FUNCTION_BLOCK M_ADD (* Add two matrices of REAL *)
  (* Standard: 61499-1 *)
  (* Version 0.2, 2007-10-24, JHC, Holobloc Inc, Changed RHS of sequences to MATRIX. *)
  (* Version 0.1, 2007-10-19, JHC, Holobloc Inc, Moved to fb.rt.math.matrix. *)
  (* Version 0.0, 2002-03-05, JHC, Rockwell Automation *)
  (* Compiler header: package fb.rt.math.matrix; *)
  (* Compiler Java Sun JDK 1.6.0 *)
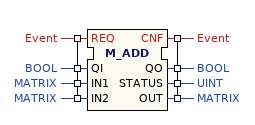
  EVENT_INPUT
    REQ WITH QI, IN1, IN2; (* Set OUT to IN1+IN2 *)
  END_EVENT
  EVENT_OUTPUT
    CNF WITH QO, STATUS, OUT; (* Confirmation of Requested Service *)
  END_EVENT
  VAR_INPUT
    QI : BOOL; (* Event Input Qualifier *)
    IN1 : MATRIX; (* Augend *)
    IN2 : MATRIX; (* Addend *)
  END_VAR
  VAR_OUTPUT
    QO : BOOL; (* Event Output Qualifier *)
    STATUS : UINT; (* Service Status *)
    OUT : MATRIX; (* Sum *)
  END_VAR
  SERVICE ADD_M/MATRIX
    SEQUENCE normal_addition
      ADD_M.REQ+(IN1,IN2) -> MATRIX.sum(IN1,IN2,OUT) -> ADD_M.CNF+(OUT);
    END_SEQUENCE
    SEQUENCE addition_inhibited
      ADD_M.REQ-() -> ADD_M.CNF-(STATUS=INHIBITED);
    END_SEQUENCE
    SEQUENCE array_size_error
      ADD_M.REQ+(IN1,IN2) -> MATRIX.sum(IN1,IN2,OUT) -> ADD_M.CNF-(STATUS=ARRAY_SIZE_ERROR);
    END_SEQUENCE
  END_SERVICE
END_FUNCTION_BLOCK
